// WC1 B1L0
TYPE ST_WP_Toilet1 :
STRUCT
	fbButton1		: FB_DigitalIn;
END_STRUCT
END_TYPE

(* stored: Version 1.1.0.1, ProductVersion 3.1.4024.12
   DUT ST_WP_Toilet1: Id {ae841982-786f-4bae-9b62-8ad9957f0e23} *)
